(* CODESYS project PROF.project

Project tree, tasks and I/O mapping:
  Device : CODESYS Control Win V3, 3S - Smart Software Solutions GmbH, order no. 305021, version 3.5.11.30
    application Application
      libraries: Standard, * (System)
      task MainTask (cyclic, interval t#20ms, priority 1) calls PLC_PRG
      task VISU_TASK (cyclic, interval 100 ms, priority 31) calls VisuElems.Visu_Prg
      program PLC_PRG [LD]
      visualisation Visualization
  text list GlobalTextList
*)

// Device/Application/PLC_PRG
PROGRAM PLC_PRG
VAR
	BOMBA   : BOOL;
	BOTAO  : BOOL;
	LIGADO : BOOL;
	PRESSAO: BOOL;
	LAMPADA: BOOL;
END_VAR

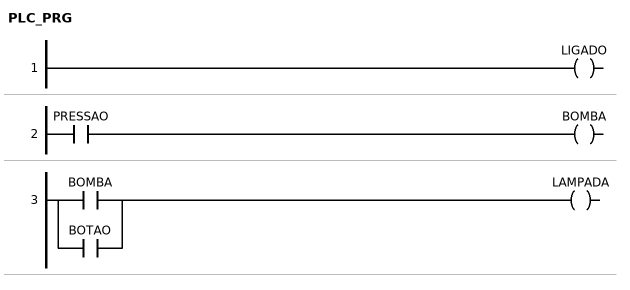
// NETWORK 1
LIGADO := TRUE;

// NETWORK 2
BOMBA := PRESSAO;

// NETWORK 3
LAMPADA := BOMBA OR BOTAO;

END_PROGRAM

// Device/Application/Visualization
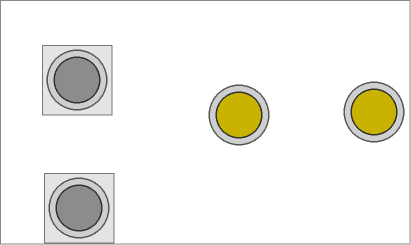
VISUALIZATION Visualization  // 411x245
    Lamp1 (204,80 70x70), variable: PLC_PRG.LAMPADA, style: Lamp-Lamp1-Yellow
    PushSwitchLed (42,45 70x70), variable: PLC_PRG.BOTAO, behaviour: TOGGLE, style: Switch-PushSwitchLed-Gray
    Lamp1 (339,77 70x70), variable: PLC_PRG.BOMBA, style: Lamp-Lamp1-Yellow
    PushSwitchLed (44,173 70x70), variable: PLC_PRG.PRESSAO, behaviour: TOGGLE, style: Switch-PushSwitchLed-Gray
END_VISUALIZATION
